{attribute 'GeneratedUsingTerminal: EL6690-0001-0000'}
{attribute addProperty BoxType "EL6690-0001-0000"}
{attribute addProperty Id "StatusAT %I*Status_D30DC33F1InputsEMPTY_STRUCTURE0OutputsEMPTY_STRUCTURE0WcStateAT %I*WcState_9091E0EB2InfoDataAT %I*InfoData_32EB74EA10"}
{attribute addProperty CRC "4245987266"}
{attribute addProperty Size "13"}
TYPE EL6690_FD149FC2 EXTENDS EtcSlaveTerminalBase_947E5A46 :
STRUCT
	{attribute addProperty Name "Status"}
	Status : Status_D30DC33F;
	{attribute addProperty Name "Inputs"}
	Inputs : EMPTY_STRUCTURE;
	{attribute addProperty Name "Outputs"}
	Outputs : EMPTY_STRUCTURE;
	{attribute addProperty Name "WcState"}
	WcState : WcState_9091E0EB;
	{attribute addProperty Name "InfoData"}
	InfoData : InfoData_32EB74EA;
END_STRUCT
END_TYPE

(* stored: Version 1.2.0.0, ProductVersion 3.1.4024.9
   DUT EL6690_FD149FC2: Id {89d81754-6df2-47be-92e3-1d5c6dd8f5dd} *)
